TYPE T_FileExtension : STRING[4];
END_TYPE

(* stored: Version 1.1.0.1
   DUT T_FileExtension: Id {09f64335-504d-4c2e-928c-25e92d302eae} *)
